{attribute 'linkalways'} 
{attribute 'no_explicit_call' := 'This FB is a CLASS and must be accessed using methods or properties'}
{attribute 'enable_dynamic_creation'}
FUNCTION_BLOCK Node_ContainerType_Vector_TcVnVector2_DINT EXTENDS Node
VAR
    out : _GUID;
END_VAR

METHOD PUBLIC  Clone : I_Node
VAR
	pNode : POINTER TO Node_ContainerType_Vector_TcVnVector2_DINT;
END_VAR
pNode := __NEW(Node_ContainerType_Vector_TcVnVector2_DINT);
Clone := pNode^;
END_METHOD

METHOD FB_init : BOOL
VAR_INPUT
	bInitRetains : BOOL; // if TRUE, the retain variables are initialized (warm start / cold start)
	bInCopyCode : BOOL;  // if TRUE, the instance afterwards gets moved into the copy code (online change)
END_VAR
AddOutput('out', out);
END_METHOD

METHOD PROTECTED OnExecute
out.Value := ContainerType_Vector_TcVnVector2_DINT;
END_METHOD

END_FUNCTION_BLOCK

(* stored: Version 1.1.0.1, ProductVersion 3.1.4026.17
   POU Node_ContainerType_Vector_TcVnVector2_DINT: Id {cb922e8e-4a56-0262-2d3e-c5d1edd28f57}, SpecialFunc None
   Folder Constructor: Id {3d8f01c6-9b7b-0d1e-036c-225e13d9b20e}
   Method Clone: Id {220ab015-54c3-0260-1cf4-943d9fc51d96}
   Method FB_init: Id {9c686311-fe62-08da-0a93-3927166ec593}
   Method OnExecute: Id {803650d1-8502-0086-0b37-4bd118c475af} *)
